// SIMATIC STEP 7 (V5.x) project Station Automatisée
// CPU: CPU 313C-2 DP
// station: Matériel
// station: SIMATIC 300(1)
// station: P_ADR_BUS
// program: Programme S7(1)

SYMBOL_TABLE
"btn dcy"	I 0.0	BOOL	// Commencer le cycle
"btn arret"	I 0.1	BOOL	// Arreter le cycle
"s1"	I 0.2	BOOL	// Detection de voiture en sortie (à l'interieur)
"s2"	I 0.3	BOOL	// Detection de voiture en sortie (à l'exterieur)
"e1"	I 0.4	BOOL	// Detection de voiture en entrée (à l'exterieur)
"e2"	I 0.5	BOOL	// Detection de voiture en entrée (à l'interieur)
"eb"	I 0.6	BOOL	// Vérin d'entrée à la position basse
"eh"	I 0.7	BOOL	// Vérin d'entrée à la position haute
"sb"	I 1.0	BOOL	// Vérin de sortie à la position basse
"sh"	I 1.1	BOOL	// Vérin de sortie à la position haute
"x0"	M 0.0	BOOL
"x1"	M 0.1	BOOL
"x100"	M 0.2	BOOL
"x101"	M 0.3	BOOL
"x102"	M 0.4	BOOL
"x103"	M 0.5	BOOL
"x200"	M 0.6	BOOL
"x201"	M 0.7	BOOL
"x202"	M 1.0	BOOL
"x203"	M 1.1	BOOL
"x300"	M 1.2	BOOL
"x301"	M 1.3	BOOL
"x302"	M 1.4	BOOL
"x400"	M 1.5	BOOL
"x401"	M 1.6	BOOL
"x402"	M 1.7	BOOL
"COMPLETE RESTART"	OB 100	OB 100	// Complete restart
"m1+"	Q 0.0	BOOL	// Avancer le vérin d'entrée
"m1-"	Q 0.1	BOOL	// Reculer le vérin d'entrée
"m2+"	Q 0.2	BOOL	// Avancer le vérin de sortie
"m2-"	Q 0.3	BOOL	// Reculer le vérin de sortie
"lev"	Q 0.4	BOOL	// Lampe d'entrée verte
"ler"	Q 0.5	BOOL	// Lampe d'entrée rouge
"lsv"	Q 0.6	BOOL	// Lampe de sortie verte
"lsr"	Q 0.7	BOOL	// Lampe de sortie rouge
END_SYMBOL_TABLE

FUNCTION FC 1 : VOID
TITLE = Grafcet d'entrée
//Traduction du grafcet d'entrée (avec une capacité max = 3)
VERSION : 0.1
BEGIN
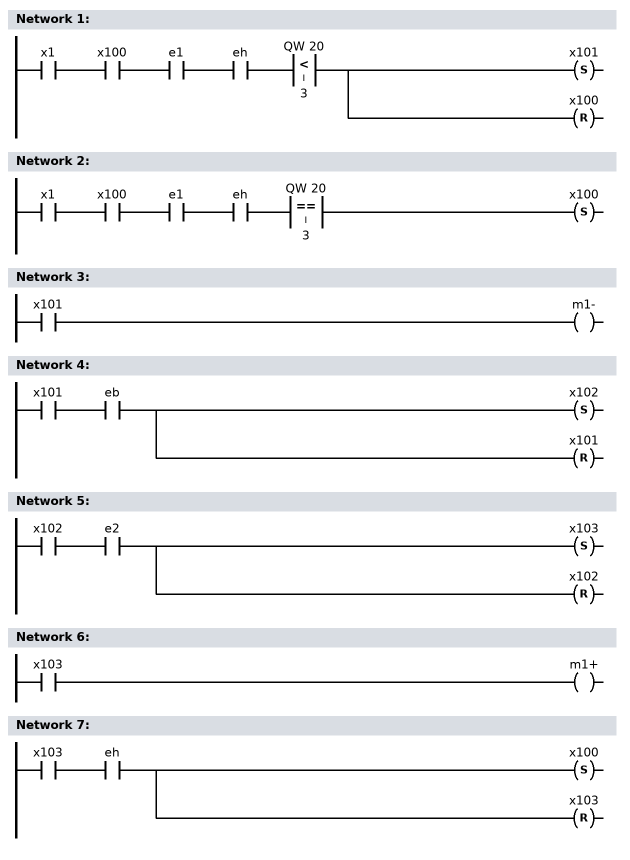
NETWORK
TITLE =
      A     "x1";
      A     "x100";
      A     "e1";
      A     "eh";
      A(;
      L     QW 20;
      L     3;
      <I;
      );
      S     "x101";
      R     "x100";
NETWORK
TITLE =
      A     "x1";
      A     "x100";
      A     "e1";
      A     "eh";
      A(;
      L     QW 20;
      L     3;
      ==I;
      );
      S     "x100";
NETWORK
TITLE =
      A     "x101";
      =     "m1-";
NETWORK
TITLE =
      A     "x101";
      A     "eb";
      S     "x102";
      R     "x101";
NETWORK
TITLE =
      A     "x102";
      A     "e2";
      S     "x103";
      R     "x102";
NETWORK
TITLE =
      A     "x103";
      =     "m1+";
NETWORK
TITLE =
      A     "x103";
      A     "eh";
      S     "x100";
      R     "x103";
END_FUNCTION

FUNCTION FC 2 : VOID
TITLE = Grafcet de sortie
//Traduction du grafcet de sortie
VERSION : 0.1
BEGIN
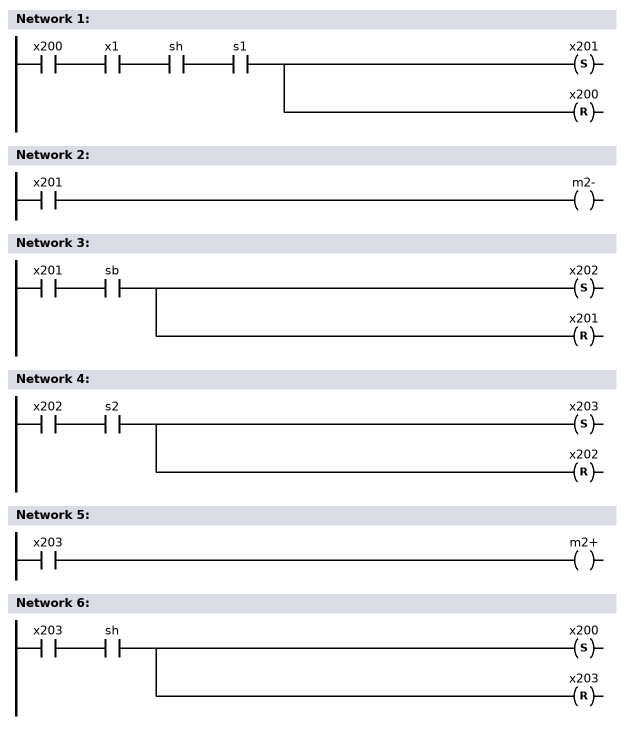
NETWORK
TITLE =
      A     "x200";
      A     "x1";
      A     "sh";
      A     "s1";
      S     "x201";
      R     "x200";
NETWORK
TITLE =
      A     "x201";
      =     "m2-";
NETWORK
TITLE =
      A     "x201";
      A     "sb";
      S     "x202";
      R     "x201";
NETWORK
TITLE =
      A     "x202";
      A     "s2";
      S     "x203";
      R     "x202";
NETWORK
TITLE =
      A     "x203";
      =     "m2+";
NETWORK
TITLE =
      A     "x203";
      A     "sh";
      S     "x200";
      R     "x203";
END_FUNCTION

FUNCTION FC 3 : VOID
TITLE = Lampe d'entrée
//Traduction du grafcet de lampe d'entrée
VERSION : 0.1
BEGIN
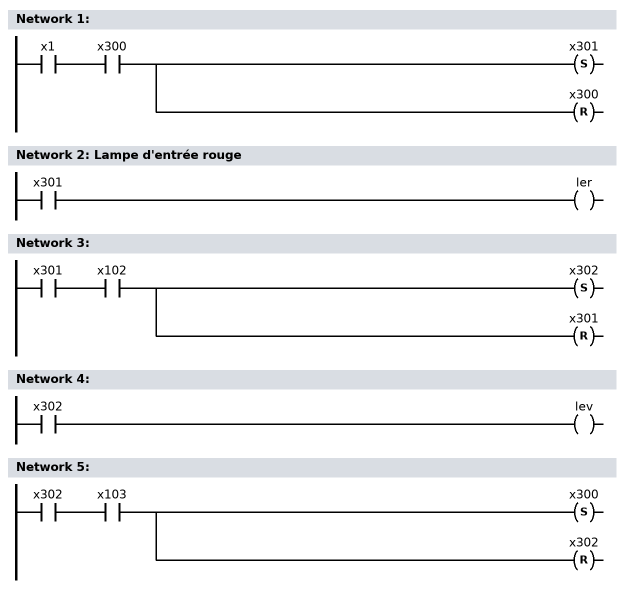
NETWORK
TITLE =
      A     "x1";
      A     "x300";
      S     "x301";
      R     "x300";
NETWORK
TITLE = Lampe d'entrée rouge
      A     "x301";
      =     "ler";
NETWORK
TITLE =
      A     "x301";
      A     "x102";
      S     "x302";
      R     "x301";
NETWORK
TITLE =
      A     "x302";
      =     "lev";
NETWORK
TITLE =
      A     "x302";
      A     "x103";
      S     "x300";
      R     "x302";
END_FUNCTION

FUNCTION FC 4 : VOID
TITLE = Lampe de sortie
//Traduction du grafcet de la lampe de sortie
//
VERSION : 0.1
BEGIN
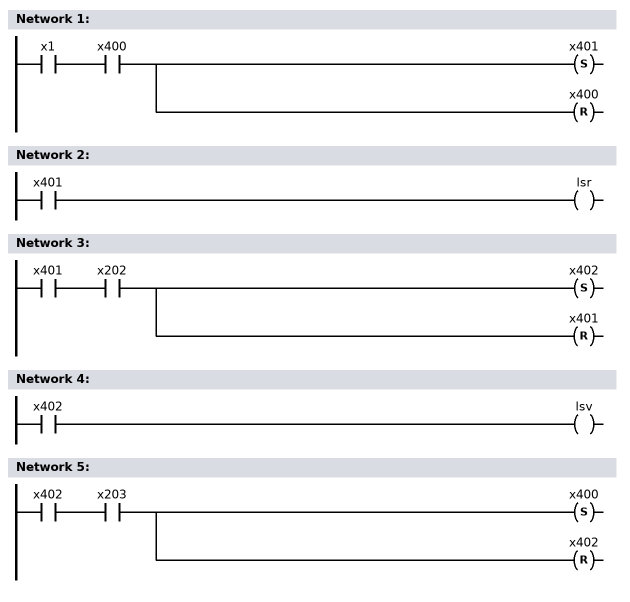
NETWORK
TITLE =
      A     "x1";
      A     "x400";
      S     "x401";
      R     "x400";
NETWORK
TITLE =
      A     "x401";
      =     "lsr";
NETWORK
TITLE =
      A     "x401";
      A     "x202";
      S     "x402";
      R     "x401";
NETWORK
TITLE =
      A     "x402";
      =     "lsv";
NETWORK
TITLE =
      A     "x402";
      A     "x203";
      S     "x400";
      R     "x402";
END_FUNCTION

FUNCTION FC 5 : VOID
TITLE = Grafcet de controle
//Traduction du grafcet de controle
VERSION : 0.1
BEGIN
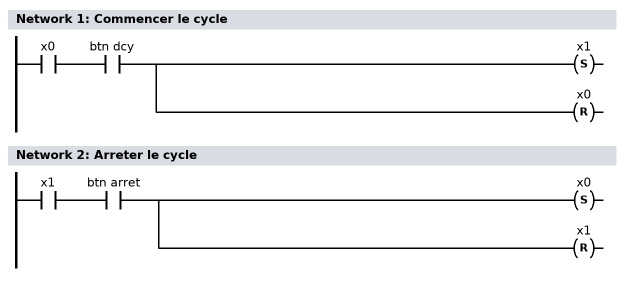
NETWORK
TITLE = Commencer le cycle
      A     "x0";
      A     "btn dcy";
      S     "x1";
      R     "x0";
NETWORK
TITLE = Arreter le cycle
      A     "x1";
      A     "btn arret";
      S     "x0";
      R     "x1";
END_FUNCTION

ORGANIZATION_BLOCK OB 1
TITLE = Main Program Sweep (Cycle)
//Programme principal: Liaison de toutes les fonctions déjà crées
VERSION : 0.1
VAR_TEMP
  OB1_EV_CLASS : BYTE ;	//Bits 0-3 = 1 (Coming event), Bits 4-7 = 1 (Event class 1)
  OB1_SCAN_1 : BYTE ;	//1 (Cold restart scan 1 of OB 1), 3 (Scan 2-n of OB 1)
  OB1_PRIORITY : BYTE ;	//Priority of OB Execution
  OB1_OB_NUMBR : BYTE ;	//1 (Organization block 1, OB1)
  OB1_RESERVED_1 : BYTE ;	//Reserved for system
  OB1_RESERVED_2 : BYTE ;	//Reserved for system
  OB1_PREV_CYCLE : INT ;	//Cycle time of previous OB1 scan (milliseconds)
  OB1_MIN_CYCLE : INT ;	//Minimum cycle time of OB1 (milliseconds)
  OB1_MAX_CYCLE : INT ;	//Maximum cycle time of OB1 (milliseconds)
  OB1_DATE_TIME : DATE_AND_TIME ;	//Date and time OB1 started
  set : BOOL ;
END_VAR
BEGIN
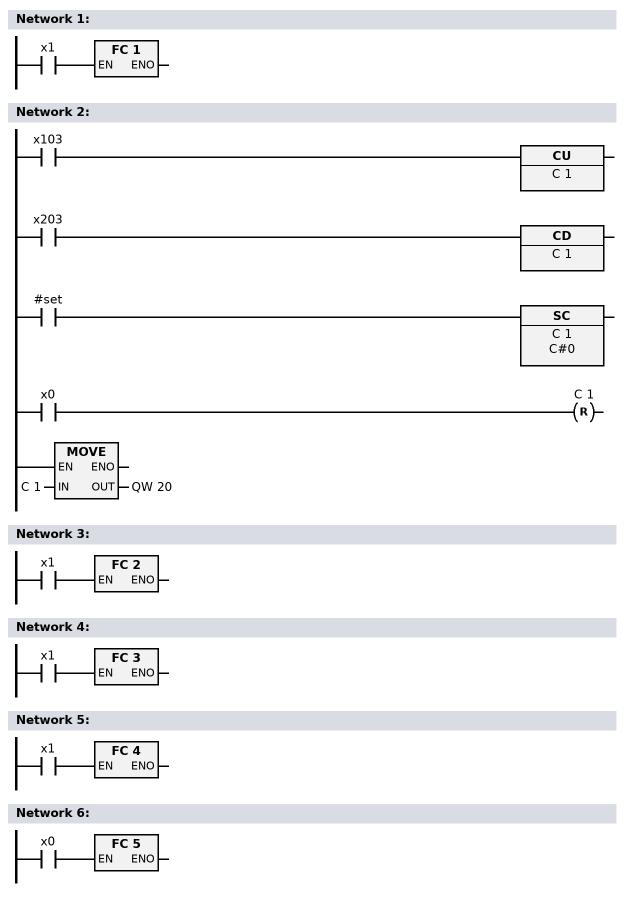
NETWORK
TITLE =
      A     "x1";
      JNB   _001;
      CALL  FC 1;
_001: NOP   0;
NETWORK
TITLE =
      A     "x103";
      CU    C 1;
      A     "x203";
      CD    C 1;
      A     #set;
      L     C#0;
      S     C 1;
      A     "x0";
      R     C 1;
      L     C 1;
      T     QW 20;
      NOP   0;
      NOP   0;
NETWORK
TITLE =
      A     "x1";
      JNB   _002;
      CALL  FC 2;
_002: NOP   0;
NETWORK
TITLE =
      A     "x1";
      JNB   _003;
      CALL  FC 3;
_003: NOP   0;
NETWORK
TITLE =
      A     "x1";
      JNB   _004;
      CALL  FC 4;
_004: NOP   0;
NETWORK
TITLE =
      A     "x0";
      JNB   _005;
      CALL  FC 5;
_005: NOP   0;
END_ORGANIZATION_BLOCK

ORGANIZATION_BLOCK "COMPLETE RESTART"	// OB 100
TITLE = Complete restart
//Initialisation du grafcet et des macro étapes
VERSION : 0.1
VAR_TEMP
  OB100_EV_CLASS : BYTE ;	//16#13, Event class 1, Entering event state, Event logged in diagnostic buffer
  OB100_STRTUP : BYTE ;	//16#81/82/83/84 Method of startup
  OB100_PRIORITY : BYTE ;	//Priority of OB Execution
  OB100_OB_NUMBR : BYTE ;	//100 (Organization block 100, OB100)
  OB100_RESERVED_1 : BYTE ;	//Reserved for system
  OB100_RESERVED_2 : BYTE ;	//Reserved for system
  OB100_STOP : WORD ;	//Event that caused CPU to stop (16#4xxx)
  OB100_STRT_INFO : DWORD ;	//Information on how system started
  OB100_DATE_TIME : DATE_AND_TIME ;	//Date and time OB100 started
END_VAR
BEGIN
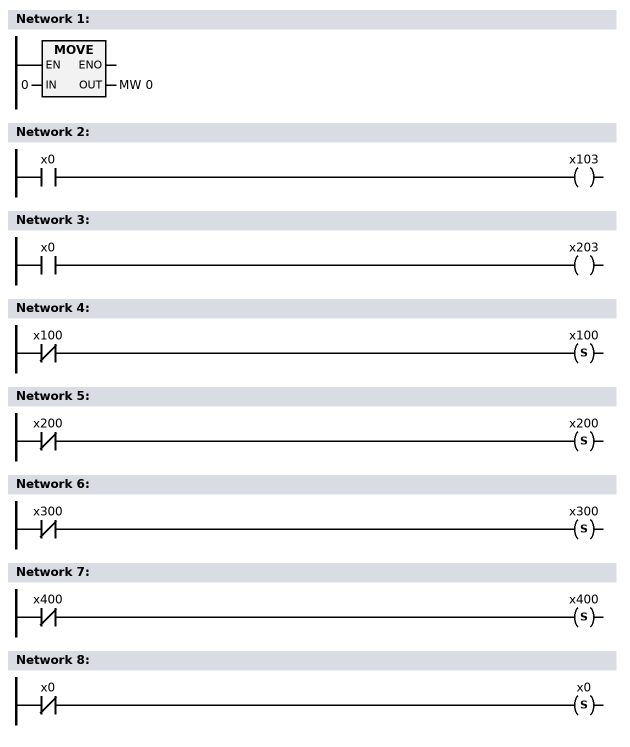
NETWORK
TITLE =
      L     0;
      T     MW 0;
      NOP   0;
NETWORK
TITLE =
      A     "x0";
      =     "x103";
NETWORK
TITLE =
      A     "x0";
      =     "x203";
NETWORK
TITLE =
      AN    "x100";
      S     "x100";
NETWORK
TITLE =
      AN    "x200";
      S     "x200";
NETWORK
TITLE =
      AN    "x300";
      S     "x300";
NETWORK
TITLE =
      AN    "x400";
      S     "x400";
NETWORK
TITLE =
      AN    "x0";
      S     "x0";
END_ORGANIZATION_BLOCK
